TYPE ST_PNOutput_PeakShaveBox :
STRUCT
	w_Status					:	WORD;
	w_Warnings					:	WORD;
	w_Faults					:	WORD;
	
	i_ActivePower				:	INT;
	i_ReactivePower				:	INT;
	ui_Frequency				:	UINT;
	ui_VoltageL1N				:	UINT;
	ui_VoltageL2N				:	UINT;
	ui_VoltageL3N				:	UINT;
	ui_VoltageL1L2				:	UINT;
	ui_VoltageL2L3				:	UINT;
	ui_VoltageL3L1				:	UINT;
	i_CurrentL1					:	INT;
	i_CurrentL2					:	INT;
	i_CurrentL3					:	INT;
	i_CurrentN					:	INT;
END_STRUCT
END_TYPE

(* stored: Version 1.1.0.1, ProductVersion 3.1.4024.12
   DUT ST_PNOutput_PeakShaveBox: Id {4662d6a3-8fa5-43c4-b929-17ce1b60f806} *)
